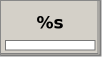
VISUALIZATION VISU_MTCSSubSystemButton  // 102x57
VAR_IN_OUT
	name : STRING;
    healthBusyStatus : HealthBusyStatusWidget;
    currentTab : STRING;
END_VAR
    Button (0,0 100x55), pressed state: currentTab = name
    Rectangle (5,40 90x10), colour variable: healthBusyStatus.bgColor
    Rectangle (0,5 100x35), "%s", text variable: name
END_VISUALIZATION

(* stored: Version 1.1.0.1, ProductVersion 3.1.0.36
   Visu VISU_MTCSSubSystemButton: Id {a2e09840-66c5-4867-97c3-85e678e47677} *)
